Omron Sysmac Studio project 1.10_marked_t1andt2_reorganised_v2 (Sysmac Studio 1.54.0.64019, StandardProject)

# Controller new_Controller_0: NJ301-1100 version 1.14
Units and slaves: Node1 : NX-ECC201 (E001); Unit 1 : NX-PC0020 (N1); Unit 2 : NX-ID5442 (N2); Unit 3 : NX-PC0010 (N3); Unit 4 : NX-PC0020 (N4); Unit 5 : NX-OD5121 (N5); Unit 6 : NX-PC0010 (N6); Power Supply : NJ-Px3001; CPU : NJ301-1100; 0 [Unit 0] : CJ1W-AD041-V1 (J01); 1 [Unit 1] : CJ1W-DA041 (J02); 2 : CJ1W-ID211 (J03); 3 : CJ1W-OC211 (J04)
Task PrimaryTask (priority 4, period or condition 1000): Program0

VAR_GLOBAL
    Station_1B2 : BOOL;  (* Ejection Cylinder Extended; at IOBus://rack#0/slot#2/Ch1_In/Ch1_In01; published *)
    Station_1B1 : BOOL;  (* Ejection Cylinder retracted; at IOBus://rack#0/slot#2/Ch1_In/Ch1_In02; published *)
    Station_2B1 : BOOL;  (* Workpiece gripped; at IOBus://rack#0/slot#2/Ch1_In/Ch1_In03; published *)
    Station_3S1 : BOOL;  (* arm_in_magazine; at IOBus://rack#0/slot#2/Ch1_In/Ch1_In04; published *)
    Station_3S2 : BOOL;  (* arm_in_downstream; at IOBus://rack#0/slot#2/Ch1_In/Ch1_In05; published *)
    Station_B4 : BOOL;  (* Magzine empty; at IOBus://rack#0/slot#2/Ch1_In/Ch1_In06; published *)
    Panel_S1 : BOOL;  (* start_button; at IOBus://rack#0/slot#2/Ch1_In/Ch1_In08; published *)
    Panel_S2 : BOOL;  (* stop_button; at IOBus://rack#0/slot#2/Ch1_In/Ch1_In09; published *)
    Panel_S4 : BOOL;  (* reset_button; at IOBus://rack#0/slot#2/Ch1_In/Ch1_In11; published *)
    Station_1Y1 : BOOL;  (* Magzine eject; at IOBus://rack#0/slot#3/Ch1_Out/Ch1_Out00; published *)
    Station_2Y1 : BOOL;  (* Vacuum on; at IOBus://rack#0/slot#3/Ch1_Out/Ch1_Out01; published *)
    Station_2Y2 : BOOL;  (* Ejector_Pulse_On; at IOBus://rack#0/slot#3/Ch1_Out/Ch1_Out02; published *)
    Station_3Y1 : BOOL;  (* arm_2_magazine; at IOBus://rack#0/slot#3/Ch1_Out/Ch1_Out03; published *)
    Station_3Y2 : BOOL;  (* arm_2_downstream; at IOBus://rack#0/slot#3/Ch1_Out/Ch1_Out04; published *)
    Station_H1 : BOOL;  (* start light; at IOBus://rack#0/slot#3/Ch1_Out/Ch1_Out08; published *)
    Station_H2 : BOOL;  (* reset light; at IOBus://rack#0/slot#3/Ch1_Out/Ch1_Out09; published *)
    Panel_H3 : BOOL;  (* Q1 light; at IOBus://rack#0/slot#3/Ch1_Out/Ch1_Out10; published *)
    Panel_H4 : BOOL;  (* Q2 light; at IOBus://rack#0/slot#3/Ch1_Out/Ch1_Out11; published *)
    Station_1B1_in : BOOL;
    IP_FI : BOOL;  (* Succeeding Station Free; at IOBus://rack#0/slot#2/Ch1_In/Ch1_In07 *)
END_VAR

PROGRAM Program0
VAR
    FB_Panel_1 : FB_Panel;
    run_mode : BOOL;
    stop_mode : BOOL;
    reset_mode : BOOL;
    FB_Actuator_T1_1 : FB_Actuator_T1;
    timer_t1 : TON;
    error_arm : BOOL;
    error_mode : BOOL;
    FB_Actuator_T2_1 : FB_Actuator_T2;
    Piston : RS;
    error_ejec : BOOL;
    extend_piston : BOOL;
    workpiece_ready_set : BOOL;
    flip_flop_1 : RS;
    workpiece_ready : BOOL;
    workpiece_picked_up : BOOL;
    wait_for_piston : TON;
    Workpiece_Checker_1 : Workpiece_Checker;
    error_state : BOOL;
    error_suction : BOOL;
    error_t1 : BOOL;
    error_t2 : BOOL;
    rs1 : RS;
    rs2 : RS;
    rs3 : RS;
    e1 : BOOL;
    e2 : BOOL;
    e3 : BOOL;
    move_to_sub : BOOL;
    vac_flipflop : RS;
    reset_vac : BOOL;
    TOF_1 : TOF;
    FB_T1_Control_1 : FB_T1_Control;
    FB_T2_Control_1 : FB_T2_Control;
    Station_H3 : BOOL;
    start_reciever : BOOL;
    stop_reciever : BOOL;
    reset_reciever : BOOL;
    next_station_ready : BOOL;
    start_button : BOOL;
    stop_button : BOOL;
    reset_button : BOOL;
    FB_Reciever_1 : FB_Receiver;
    Workpeice_Checker_2_next_station : Workpiece_Checker;
    next_station_ready_set : BOOL;
    test_next_station_rs : RS;
    next_station_ready_check_1 : next_station_ready_check;
    next_station_free_in : BOOL;
END_VAR
VAR_EXTERNAL
    Station_3S1 : BOOL;
    Panel_S2 : BOOL;
    Station_3Y2 : BOOL;
    Station_3S2 : BOOL;
    Panel_S1 : BOOL;
    Station_3Y1 : BOOL;
    Panel_S4 : BOOL;
    Station_H1 : BOOL;
    Station_H2 : BOOL;
    Panel_H4 : BOOL;
    Panel_H3 : BOOL;
    Station_1B2 : BOOL;
    Station_1B1 : BOOL;
    Station_1Y1 : BOOL;
    Station_2Y1 : BOOL;
    Station_2B1 : BOOL;
    Station_B4 : BOOL;
    Station_2Y2 : BOOL;
    IP_FI : BOOL;
END_VAR
VAR
    _e1 : F_TRIG;
    _e2 : F_TRIG;
END_VAR

(* Section Section0: ladder, written here as Structured Text *)

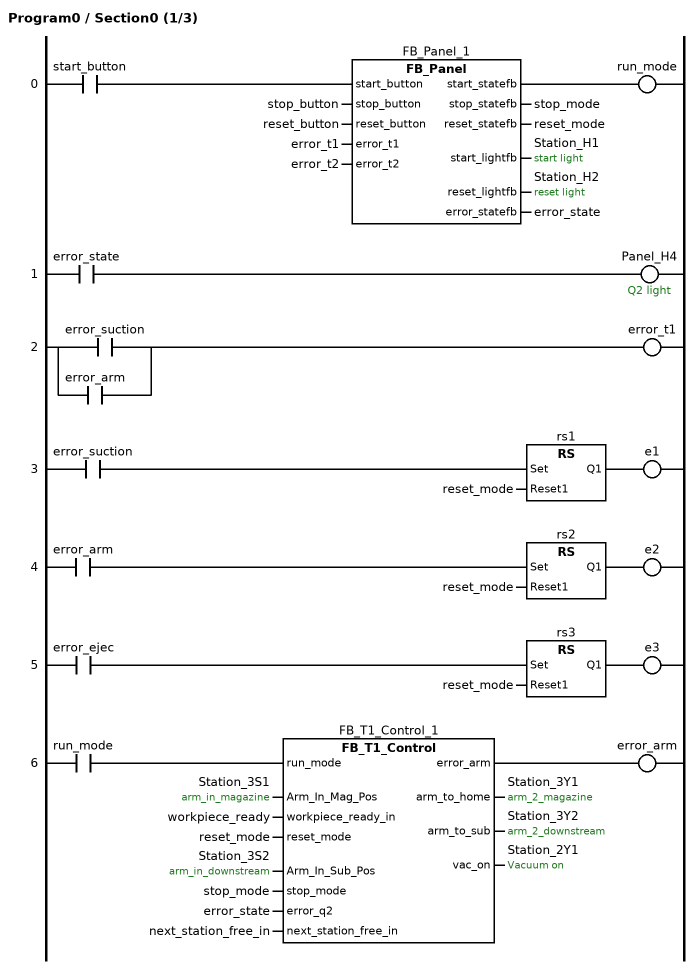
(* Rung 0 *)
FB_Panel_1(start_button := start_button, stop_button := stop_button, reset_button := reset_button, error_t1 := error_t1, error_t2 := error_t2, stop_statefb => stop_mode, reset_statefb => reset_mode, start_lightfb => Station_H1, reset_lightfb => Station_H2, error_statefb => error_state);
run_mode := FB_Panel_1.start_statefb;
(* Rung 1 *)
Panel_H4 := error_state;
(* Rung 2 *)
error_t1 := error_suction OR error_arm;
(* Rung 3 *)
rs1(Set := error_suction, Reset1 := reset_mode);
e1 := rs1.Q1;
(* Rung 4 *)
rs2(Set := error_arm, Reset1 := reset_mode);
e2 := rs2.Q1;
(* Rung 5 *)
rs3(Set := error_ejec, Reset1 := reset_mode);
e3 := rs3.Q1;
(* Rung 6 *)
FB_T1_Control_1(run_mode := run_mode, Arm_In_Mag_Pos := Station_3S1, workpiece_ready_in := workpiece_ready, reset_mode := reset_mode, Arm_In_Sub_Pos := Station_3S2, stop_mode := stop_mode, error_q2 := error_state, next_station_free_in := next_station_free_in, arm_to_home => Station_3Y1, arm_to_sub => Station_3Y2, vac_on => Station_2Y1);
error_arm := FB_T1_Control_1.error_arm;

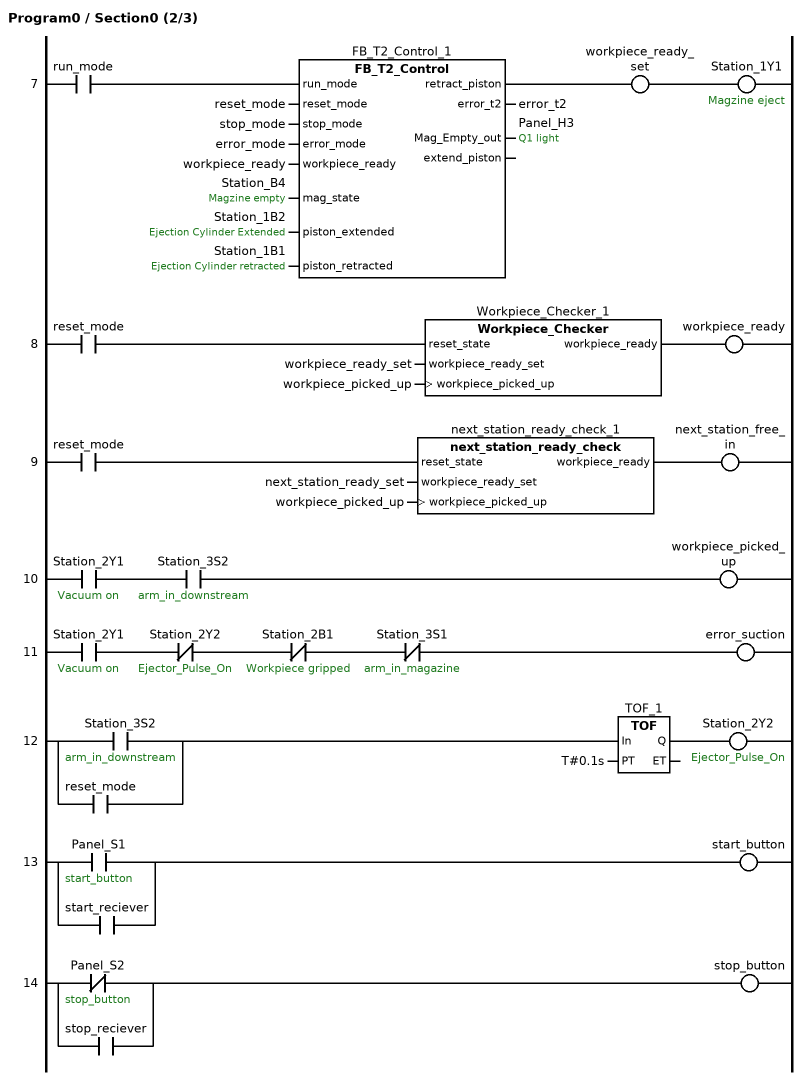
(* Rung 7 *)
FB_T2_Control_1(run_mode := run_mode, reset_mode := reset_mode, stop_mode := stop_mode, error_mode := error_mode, workpiece_ready := workpiece_ready, mag_state := Station_B4, piston_extended := Station_1B2, piston_retracted := Station_1B1, error_t2 => error_t2, Mag_Empty_out => Panel_H3);
workpiece_ready_set := FB_T2_Control_1.retract_piston;
Station_1Y1 := FB_T2_Control_1.retract_piston;
(* Rung 8 *)
_e1(CLK := workpiece_picked_up);
Workpiece_Checker_1(reset_state := reset_mode, workpiece_ready_set := workpiece_ready_set, workpiece_picked_up := _e1.Q);
workpiece_ready := Workpiece_Checker_1.workpiece_ready;
(* Rung 9 *)
_e2(CLK := workpiece_picked_up);
next_station_ready_check_1(reset_state := reset_mode, workpiece_ready_set := next_station_ready_set, workpiece_picked_up := _e2.Q);
next_station_free_in := next_station_ready_check_1.workpiece_ready;
(* Rung 10 *)
workpiece_picked_up := Station_2Y1 AND Station_3S2;
(* Rung 11 *)
error_suction := Station_2Y1 AND NOT Station_2Y2 AND NOT Station_2B1 AND NOT Station_3S1;
(* Rung 12 *)
TOF_1(In := Station_3S2 OR reset_mode, PT := T#0.1s);
Station_2Y2 := TOF_1.Q;
(* Rung 13 *)
start_button := Panel_S1 OR start_reciever;
(* Rung 14 *)
stop_button := NOT Panel_S2 OR stop_reciever;

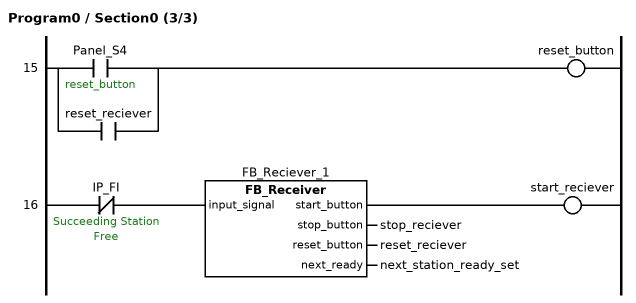
(* Rung 15 *)
reset_button := Panel_S4 OR reset_reciever;
(* Rung 16 *)
FB_Reciever_1(input_signal := NOT IP_FI, stop_button => stop_reciever, reset_button => reset_reciever, next_ready => next_station_ready_set);
start_reciever := FB_Reciever_1.start_button;
END_PROGRAM

FUNCTION_BLOCK FB_Panel
VAR
    flip_flop : RS;
    flip_flop2 : RS;
    flip_flop_3 : RS;
    flip_flop3 : RS;
    stop_or_error : BOOL;
    error_q2 : BOOL;
    flip_flop4 : RS;
END_VAR
VAR_OUTPUT
    start_statefb : BOOL;
    stop_statefb : BOOL;
    reset_statefb : BOOL;
END_VAR
VAR_INPUT
    start_button : BOOL := False;
    stop_button : BOOL := False;
    reset_button : BOOL := False;
END_VAR
VAR_OUTPUT
    start_lightfb : BOOL;
    reset_lightfb : BOOL;
    error_statefb : BOOL;
END_VAR
VAR_INPUT
    error_t1 : BOOL;
    error_t2 : BOOL;
END_VAR
VAR_EXTERNAL
    Panel_H4 : BOOL;
END_VAR
(* ladder, written here as Structured Text *)

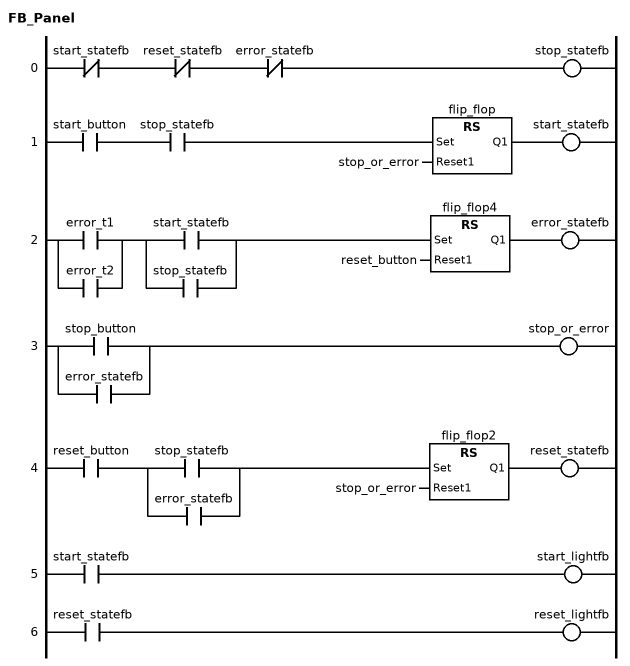
(* Rung 0 *)
stop_statefb := NOT start_statefb AND NOT reset_statefb AND NOT error_statefb;
(* Rung 1 *)
flip_flop(Set := start_button AND stop_statefb, Reset1 := stop_or_error);
start_statefb := flip_flop.Q1;
(* Rung 2 *)
flip_flop4(Set := (error_t1 OR error_t2) AND (start_statefb OR stop_statefb), Reset1 := reset_button);
error_statefb := flip_flop4.Q1;
(* Rung 3 *)
stop_or_error := stop_button OR error_statefb;
(* Rung 4 *)
flip_flop2(Set := reset_button AND (stop_statefb OR error_statefb), Reset1 := stop_or_error);
reset_statefb := flip_flop2.Q1;
(* Rung 5 *)
start_lightfb := start_statefb;
(* Rung 6 *)
reset_lightfb := reset_statefb;
END_FUNCTION_BLOCK

FUNCTION_BLOCK FB_Actuator_T1
VAR
    flip_flop_1 : RS;
    flip_flop_2 : RS;
    reset_to_home : BOOL;
    timer_t1 : TON;
    flip_flop_3 : RS;
    timer_t2 : TON;
    flip_flop_4 : RS;
    error_toSub : BOOL;
    error_toHome : BOOL;
    middle_timer : AccumulationTimer;
    flip_flop_5 : RS;
    reset_middle : BOOL;
    flip_flop6 : RS;
    move_to_middle_from_home : BOOL;
    move_to_home : BOOL;
    move_to_middle_from_sub : BOOL;
    unknown_pos : BOOL;
    reset_vac_arm_to_sub : BOOL;
    timer_t3 : TON;
    t : TIME;
    unknown_pos_timer : TON;
    TOF_1 : TOF;
    move_to_sub : BOOL;
    rese : BOOL;
END_VAR
VAR_INPUT
    Arm_In_Mag_Pos : BOOL;
    Arm_In_Sub_Pos : BOOL;
    stop_mode : BOOL;
END_VAR
VAR_OUTPUT
    error_arm : BOOL;
    arm_to_sub : BOOL;
    arm_to_home : BOOL;
END_VAR
VAR_INPUT
    error_q2 : BOOL;
    set_move_to_sub : BOOL;
    set_move_to_home : BOOL;
    set_move_to_middle_from_home : BOOL;
    set_move_to_middle_from_sub : BOOL;
END_VAR
VAR_OUTPUT
    middle_pos : BOOL;
END_VAR
VAR_INPUT
    reset_mode : BOOL;
END_VAR
VAR_EXTERNAL
    Station_3S1 : BOOL;
    Station_3Y1 : BOOL;
    Station_3S2 : BOOL;
    Station_3Y2 : BOOL;
    Station_2Y2 : BOOL;
    Station_2Y1 : BOOL;
END_VAR
(* ladder, written here as Structured Text *)

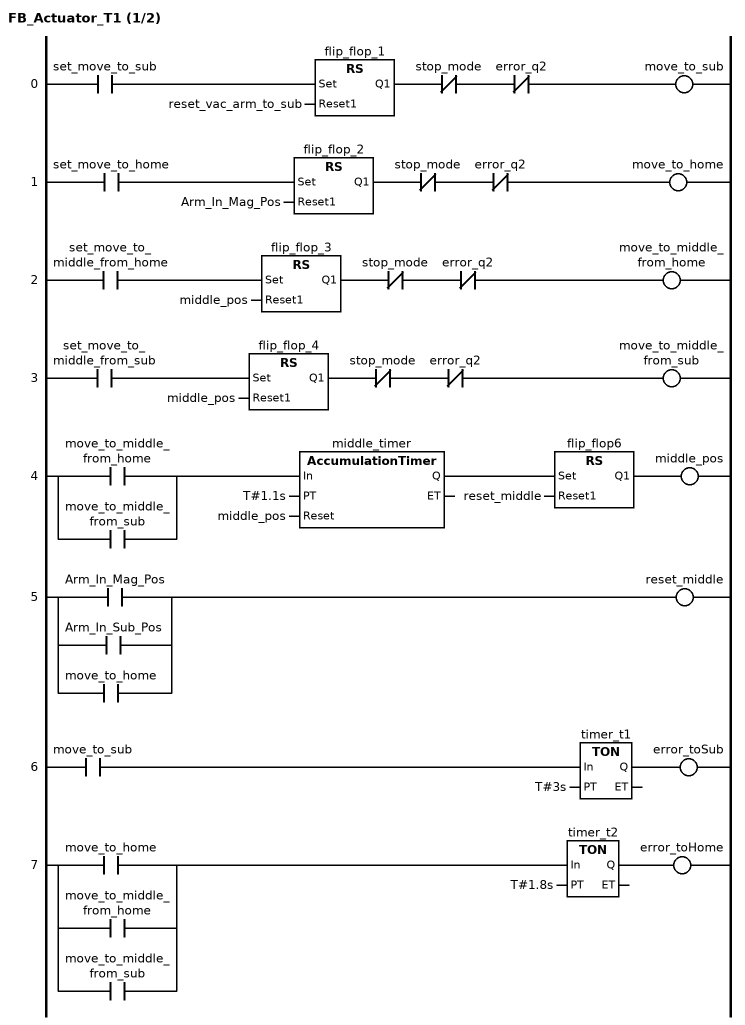
(* Rung 0 *)
flip_flop_1(Set := set_move_to_sub, Reset1 := reset_vac_arm_to_sub);
move_to_sub := flip_flop_1.Q1 AND NOT stop_mode AND NOT error_q2;
(* Rung 1 *)
flip_flop_2(Set := set_move_to_home, Reset1 := Arm_In_Mag_Pos);
move_to_home := flip_flop_2.Q1 AND NOT stop_mode AND NOT error_q2;
(* Rung 2 *)
flip_flop_3(Set := set_move_to_middle_from_home, Reset1 := middle_pos);
move_to_middle_from_home := flip_flop_3.Q1 AND NOT stop_mode AND NOT error_q2;
(* Rung 3 *)
flip_flop_4(Set := set_move_to_middle_from_sub, Reset1 := middle_pos);
move_to_middle_from_sub := flip_flop_4.Q1 AND NOT stop_mode AND NOT error_q2;
(* Rung 4 *)
middle_timer(In := move_to_middle_from_home OR move_to_middle_from_sub, PT := T#1.1s, Reset := middle_pos);
flip_flop6(Set := middle_timer.Q, Reset1 := reset_middle);
middle_pos := flip_flop6.Q1;
(* Rung 5 *)
reset_middle := Arm_In_Mag_Pos OR Arm_In_Sub_Pos OR move_to_home;
(* Rung 6 *)
timer_t1(In := move_to_sub, PT := T#3s);
error_toSub := timer_t1.Q;
(* Rung 7 *)
timer_t2(In := move_to_home OR move_to_middle_from_home OR move_to_middle_from_sub, PT := T#1.8s);
error_toHome := timer_t2.Q;

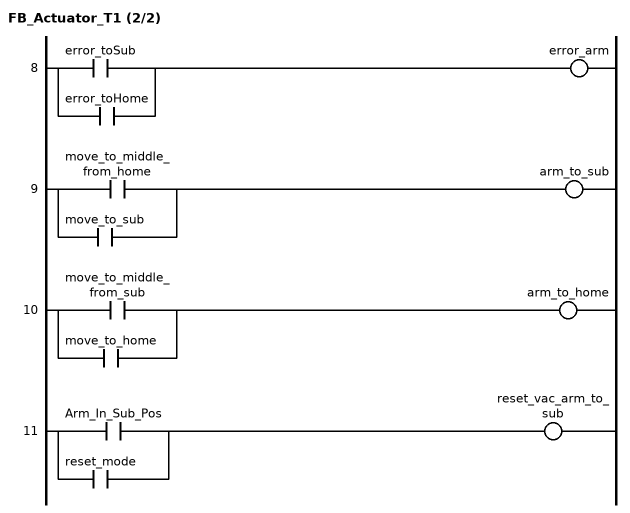
(* Rung 8 *)
error_arm := error_toSub OR error_toHome;
(* Rung 9 *)
arm_to_sub := move_to_middle_from_home OR move_to_sub;
(* Rung 10 *)
arm_to_home := move_to_middle_from_sub OR move_to_home;
(* Rung 11 *)
reset_vac_arm_to_sub := Arm_In_Sub_Pos OR reset_mode;
END_FUNCTION_BLOCK

FUNCTION_BLOCK FB_Actuator_T2
VAR
    reset_to_home : BOOL;
    retract_ff : RS;
    extend_ff : RS;
    extend_t : TON;
    retract_t : TON;
    retract_err : BOOL;
    extend_err : BOOL;
    workpiece_lifted : BOOL;
    Workpiece_ejection : RS;
END_VAR
VAR_OUTPUT
    retract_piston : BOOL;
END_VAR
VAR_INPUT
    error_mode : BOOL;
END_VAR
VAR_OUTPUT
    extend_piston : BOOL;
END_VAR
VAR_INPUT
    piston_retracted : BOOL;
    piston_extended : BOOL;
END_VAR
VAR_OUTPUT
    error_eject : BOOL;
END_VAR
VAR_INPUT
    extend_piston_command : BOOL;
    retract_piston_command : BOOL;
END_VAR
VAR_EXTERNAL
    Station_B4 : BOOL;
    Station_1B1 : BOOL;
    Station_1B2 : BOOL;
    Station_2Y1 : BOOL;
END_VAR
(* ladder, written here as Structured Text *)

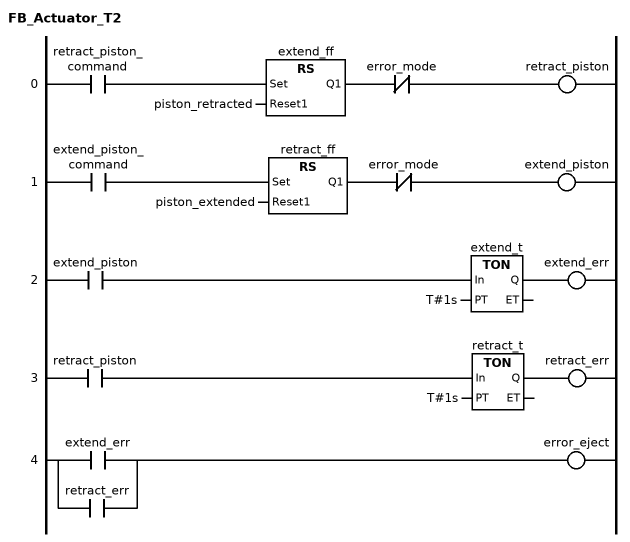
(* Rung 0 *)
extend_ff(Set := retract_piston_command, Reset1 := piston_retracted);
retract_piston := extend_ff.Q1 AND NOT error_mode;
(* Rung 1 *)
retract_ff(Set := extend_piston_command, Reset1 := piston_extended);
extend_piston := retract_ff.Q1 AND NOT error_mode;
(* Rung 2 *)
extend_t(In := extend_piston, PT := T#1s);
extend_err := extend_t.Q;
(* Rung 3 *)
retract_t(In := retract_piston, PT := T#1s);
retract_err := retract_t.Q;
(* Rung 4 *)
error_eject := extend_err OR retract_err;
END_FUNCTION_BLOCK

FUNCTION_BLOCK Workpiece_Checker
VAR
    wait_for_piston : TON;
    flip_flop_1 : RS;
    workpiece_not_ready : BOOL;
END_VAR
VAR_INPUT
    reset_state : BOOL;
    workpiece_ready_set : BOOL;
    workpiece_picked_up : BOOL (* edge DownDirection *);
END_VAR
VAR_OUTPUT
    workpiece_ready : BOOL;
END_VAR
(* ladder, written here as Structured Text *)

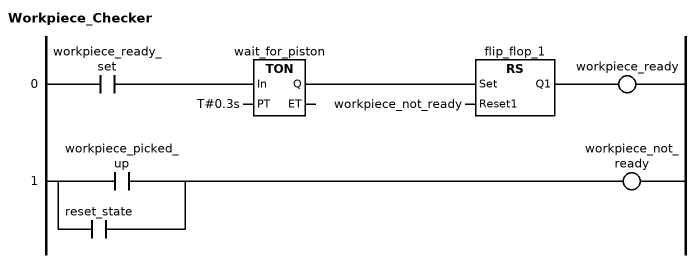
(* Rung 0 *)
wait_for_piston(In := workpiece_ready_set, PT := T#0.3s);
flip_flop_1(Set := wait_for_piston.Q, Reset1 := workpiece_not_ready);
workpiece_ready := flip_flop_1.Q1;
(* Rung 1 *)
workpiece_not_ready := workpiece_picked_up OR reset_state;
END_FUNCTION_BLOCK

FUNCTION_BLOCK FB_T1_Control
VAR
    unknown_pos : BOOL;
    unknown_pos_timer : TON;
    move_to_sub : BOOL;
    move_to_home : BOOL;
    middle_pos : BOOL;
    move_to_middle_from_home : BOOL;
    move_to_middle_from_sub : BOOL;
    FB_Actuator_T1_1 : FB_Actuator_T1;
    vac_flipflop : RS;
    reset_vac : BOOL;
END_VAR
VAR_INPUT
    run_mode : BOOL;
    Arm_In_Mag_Pos : BOOL;
    workpiece_ready_in : BOOL;
    reset_mode : BOOL;
    Arm_In_Sub_Pos : BOOL;
    stop_mode : BOOL;
END_VAR
VAR_OUTPUT
    error_arm : BOOL;
    arm_to_home : BOOL;
    arm_to_sub : BOOL;
    vac_on : BOOL;
END_VAR
VAR_INPUT
    error_q2 : BOOL;
    next_station_free_in : BOOL;
END_VAR
(* ladder, written here as Structured Text *)

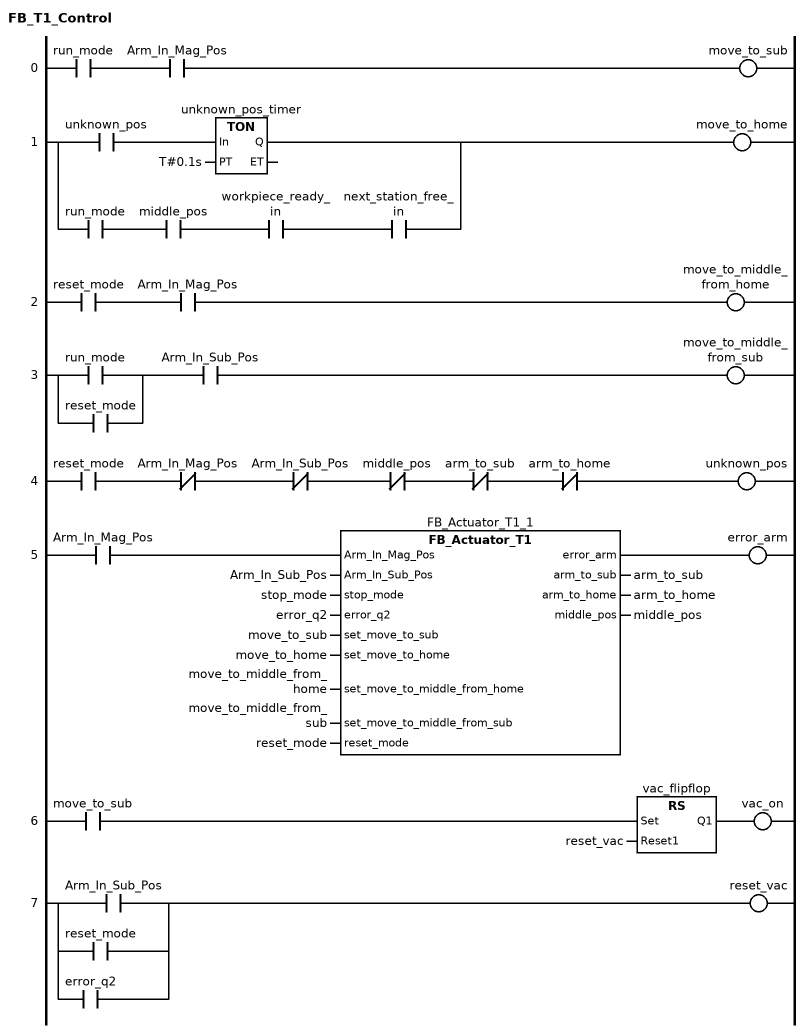
(* Rung 0 *)
move_to_sub := run_mode AND Arm_In_Mag_Pos;
(* Rung 1 *)
unknown_pos_timer(In := unknown_pos, PT := T#0.1s);
move_to_home := unknown_pos_timer.Q OR (run_mode AND middle_pos AND workpiece_ready_in AND next_station_free_in);
(* Rung 2 *)
move_to_middle_from_home := reset_mode AND Arm_In_Mag_Pos;
(* Rung 3 *)
move_to_middle_from_sub := (run_mode OR reset_mode) AND Arm_In_Sub_Pos;
(* Rung 4 *)
unknown_pos := reset_mode AND NOT Arm_In_Mag_Pos AND NOT Arm_In_Sub_Pos AND NOT middle_pos AND NOT arm_to_sub AND NOT arm_to_home;
(* Rung 5 *)
FB_Actuator_T1_1(Arm_In_Mag_Pos := Arm_In_Mag_Pos, Arm_In_Sub_Pos := Arm_In_Sub_Pos, stop_mode := stop_mode, error_q2 := error_q2, set_move_to_sub := move_to_sub, set_move_to_home := move_to_home, set_move_to_middle_from_home := move_to_middle_from_home, set_move_to_middle_from_sub := move_to_middle_from_sub, reset_mode := reset_mode, arm_to_sub => arm_to_sub, arm_to_home => arm_to_home, middle_pos => middle_pos);
error_arm := FB_Actuator_T1_1.error_arm;
(* Rung 6 *)
vac_flipflop(Set := move_to_sub, Reset1 := reset_vac);
vac_on := vac_flipflop.Q1;
(* Rung 7 *)
reset_vac := Arm_In_Sub_Pos OR reset_mode OR error_q2;
END_FUNCTION_BLOCK

FUNCTION_BLOCK FB_T2_Control
VAR
    retract_piston_command : BOOL;
    FB_Actuator_T2_1 : FB_Actuator_T2;
    extend_piston_command : BOOL;
END_VAR
VAR_INPUT
    run_mode : BOOL;
    reset_mode : BOOL;
    stop_mode : BOOL;
    error_mode : BOOL;
    workpiece_ready : BOOL;
    mag_state : BOOL;
    piston_extended : BOOL;
    piston_retracted : BOOL;
END_VAR
VAR_OUTPUT
    retract_piston : BOOL;
    error_t2 : BOOL;
    Mag_Empty_out : BOOL;
    extend_piston : BOOL;
END_VAR
(* ladder, written here as Structured Text *)

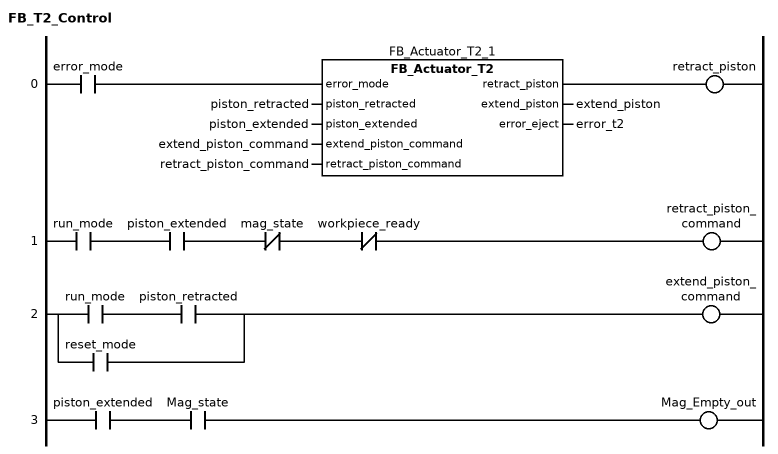
(* Rung 0 *)
FB_Actuator_T2_1(error_mode := error_mode, piston_retracted := piston_retracted, piston_extended := piston_extended, extend_piston_command := extend_piston_command, retract_piston_command := retract_piston_command, extend_piston => extend_piston, error_eject => error_t2);
retract_piston := FB_Actuator_T2_1.retract_piston;
(* Rung 1 *)
retract_piston_command := run_mode AND piston_extended AND NOT mag_state AND NOT workpiece_ready;
(* Rung 2 *)
extend_piston_command := (run_mode AND piston_retracted) OR reset_mode;
(* Rung 3 *)
Mag_Empty_out := piston_extended AND Mag_state;
END_FUNCTION_BLOCK

FUNCTION_BLOCK FB_Receiver
VAR
    pulse_length_timer : AccumulationTimer;
    reset_length : BOOL;
    pulse_length : TIME;
    timer_maxed : BOOL;
    wait_max_time : TON;
    max_time_signal : BOOL;
    start_counting_RS : RS;
    elapsed_time : TIME;
    pulse_length_comparison : FB_Reciever_Ladder_Logic;
    panel : BOOL;
    next_ready_check : RS;
END_VAR
VAR_OUTPUT
    start_button : BOOL;
    stop_button : BOOL;
    reset_button : BOOL;
    next_ready : BOOL;
END_VAR
VAR_INPUT
    input_signal : BOOL;
END_VAR
VAR_EXTERNAL
    Panel_H4 : BOOL;
    Panel_S2 : BOOL;
    Station_H2 : BOOL;
    Panel_S4 : BOOL;
END_VAR
(* ladder, written here as Structured Text *)

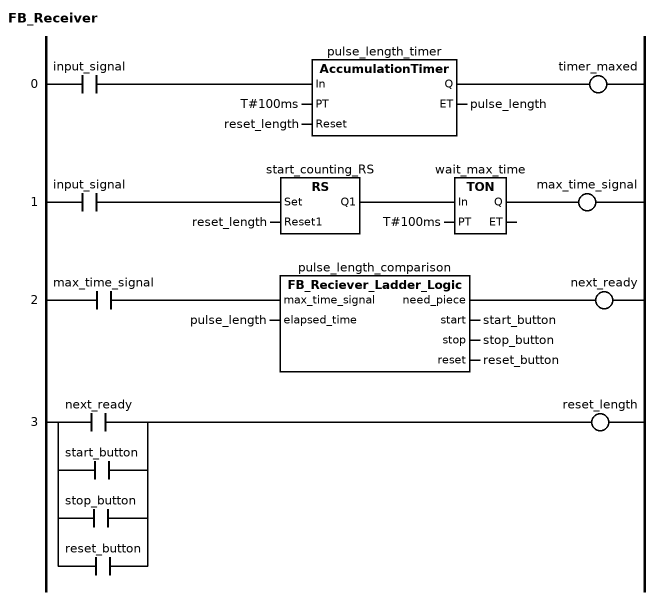
(* Rung 0 *)
pulse_length_timer(In := input_signal, PT := T#100ms, Reset := reset_length, ET => pulse_length);
timer_maxed := pulse_length_timer.Q;
(* Rung 1 *)
start_counting_RS(Set := input_signal, Reset1 := reset_length);
wait_max_time(In := start_counting_RS.Q1, PT := T#100ms);
max_time_signal := wait_max_time.Q;
(* Rung 2 *)
pulse_length_comparison(max_time_signal := max_time_signal, elapsed_time := pulse_length, start => start_button, stop => stop_button, reset => reset_button);
next_ready := pulse_length_comparison.need_piece;
(* Rung 3 *)
reset_length := next_ready OR start_button OR stop_button OR reset_button;
END_FUNCTION_BLOCK

FUNCTION_BLOCK FB_Reciever_Ladder_Logic
VAR_INPUT
    elapsed_time : TIME;
    max_time_signal : BOOL;
END_VAR
VAR_OUTPUT
    need_piece : BOOL;
    start : BOOL;
    stop : BOOL;
    reset : BOOL;
END_VAR
IF (max_time_signal) & (elapsed_time > T#70ms) THEN
	need_piece := TRUE;
	start := FALSE;
	stop := FALSE;
	reset := FALSE;
	
ELSIF (max_time_signal) & (elapsed_time > T#50ms)  THEN
	need_piece := FALSE;
	start := FALSE;
	stop := FALSE;
	reset := TRUE;

ELSIF (max_time_signal) & (elapsed_time > T#30ms)  THEN
	need_piece := FALSE;
	start := FALSE;
	stop := TRUE;
	reset := FALSE;
	
ELSIF (max_time_signal) & (elapsed_time >= T#0ms) THEN
	need_piece := FALSE;
	start := TRUE;
	stop := FALSE;
	reset := FALSE;
ELSE
	need_piece := FALSE;
	start := FALSE;
	stop := FALSE;
	reset := FALSE;

END_IF;
	
END_FUNCTION_BLOCK

FUNCTION_BLOCK next_station_ready_check
VAR
    wait_for_piston : TON;
    flip_flop_1 : RS;
    workpiece_not_ready : BOOL;
END_VAR
VAR_INPUT
    reset_state : BOOL;
    workpiece_ready_set : BOOL;
    workpiece_picked_up : BOOL (* edge DownDirection *);
END_VAR
VAR_OUTPUT
    workpiece_ready : BOOL;
END_VAR
(* ladder, written here as Structured Text *)

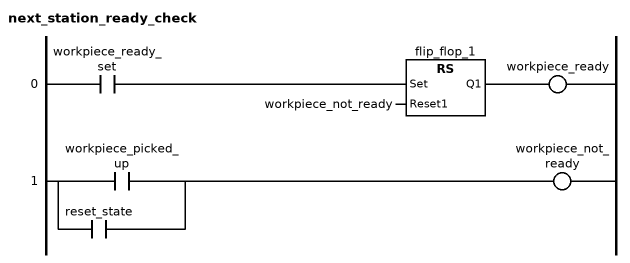
(* Rung 0 *)
flip_flop_1(Set := workpiece_ready_set, Reset1 := workpiece_not_ready);
workpiece_ready := flip_flop_1.Q1;
(* Rung 1 *)
workpiece_not_ready := workpiece_picked_up OR reset_state;
END_FUNCTION_BLOCK